{attribute 'Tc2GvlVarNames'}
{attribute 'strict'}
//Verso del Pallettizzatore
TYPE e_Verso_Pallettizzatore :
(
	PALLETTIZZATORE_DX := 1, //Identifica il pallettizzatore la cui linea di trasporti rimane ALLE SPALLE e A DESTRA
	PALLETTIZZATORE_SX := 2 //Identifica il pallettizzatore la cui linea di trasporti rimane ALLE SPALLE e A SINISTRA
);
END_TYPE

(* stored: Version 1.1.0.1, ProductVersion 3.1.4024.11
   EnumerationTextList e_Verso_Pallettizzatore: Id {2cb9d178-1f67-4ca5-b209-35229359267b} *)
